// TIA Portal V19 export
FUNCTION "CIP_Filler_512" : Void   // FC98, STL
TITLE = CIP OF FILLING MACHINE
{ S7_Optimized_Access := 'TRUE' }
NAME : CIPTANK
VERSION : 0.0
// Setpoint for Cip forward changed to real from integer
// 
// CIP Program 1 = Rinse-caustic-rinse-acid-rinse-drain
// CIP Program 2 = rinse=caustic-rinse-drain
// 
// If the combi 512 is in fault, the CIP_PUMP_ON input is false, thus M0139 is
// de-engerised and the sequence is held. When the sequence is held steam and 
// chemical valves are de-engerised.
// 
// Version 15 - 25/1/13 ...AFL
// Reset of "M_CAUSTIC_READY" ,"M_RINSE_READY", "M_ACID_READY", in step 1 after 
// occurence of CIP going through without dosing any caustic into CIP solution.
// 
// Version 16 - 22/02/13 ...MC
// In addition to above comment, "CT_LYE_OK", "CT_ACID_OK" also reset in same 
// step.
// stored: AutoNumber false
   VAR_TEMP
      RinseCount : Int;
      Count : Int;
      TEMP0 : Real;
      TEMP2 : Real;
   END_VAR
BEGIN

NETWORK
TITLE = CIP FILLING MACHINE
// Comment
// 
// 
//  Productline being cleaned - Q21.5
      A     "S0 CIP TANK";
      =     "ProdLineBeingCleaned";

// CIP Release - Q21.7
      A     "FS01.81";  // Return flow switch
      A     "Request CIP Pump ON";  //If CIP_PUMP_ON is false
      A(;
      O     "M_CAUSTIC_READY";  //reset CIP release signal
      O     "M_RINSE_READY";
      O     "M_ACID_READY";
      );
      O(;
      A     "Filler_CIP_512_DB".Drain_Ready;  // drain
      A     "Request Drain";
      );
      =     "M_CIP Release";

//   Time Stop - Q21.6
// If a FB error exists sent time stop signal to combi 512
      O     "ItemAlarmsOP".Item[9];  //FB_FAULT_VALVE_01_15
      O     "ItemAlarmsOP".Item[10];  //FB_FAULT_MOTOR_01_39
//  O     "ItemAlarmsOP".FB_FAULT_MOTOR_01_30
      O     "ItemAlarmsOP".Item[12];  //FB_FAULT_VALVE_02_37
      O     "ItemAlarmsOP".Item[13];  //FB_FAULT_VALVE_02_38
      O     "ItemAlarmsOP".Item[14];  //FB_FAULT_VALVE_01_16
      O     "ItemAlarmsOP".Item[15];  //FB_FAULT_VALVE_01_17
//   O     "ItemAlarmsOP".FB_FAULT_VALVE_01_08
//   O     "ItemAlarmsOP".FB_FAULT_VALVE_01_01
//   O     "ItemAlarmsOP".FB_FAULT_VALVE_01_03
//    O     "ItemAlarmsOP".FB_FAULT_VALVE_01_04
//      O     "ItemAlarmsOP".FB_FAULT_VALVE_01_09
//   O     "ItemAlarmsOP".FB_FAULT_VALVE_01_11
      O     "ItemAlarmsOP".Item[6];  //FB_FAULT_VALVE_01_12
      O     "ItemAlarmsOP".Item[7];  //FB_FAULT_VALVE_01_13
      O     "ItemAlarmsOP".Item[8];  //FB_FAULT_VALVE_01_14

//      O     "ItemAlarmsOP".FB_FAULT_VALVE_09_10
//      O     "ItemAlarmsOP".FB_FAULT_VALVE_09_11
//     O     "ItemAlarmsOP".FB_FAULT_VALVE_09_12

//      O     "ItemAlarmsOP".FB_FAULT_VALVE_01_19
      O     "ItemAlarmsOP".Item[18];  //FB_FAULT_VALVE_WATERPUMP
//    O     "ItemAlarmsOP".FB_FAULT_VALVE_09_04
//    O     "ItemAlarmsOP".FB_FAULT_VALVE_09_05
//    O     "ItemAlarmsOP".FB_FAULT_VALVE_09_06
//    O     "ItemAlarmsOP".FB_FAULT_VALVE_09_07
//    O     "ItemAlarmsOP".FB_FAULT_VALVE_09_08
//     O     "ItemAlarmsOP".FB_FAULT_VALVE_09_09
//      =     "M_Time Stop CIP"

      A     "S0 FILLER";
      A     "Combi 512 In USE";
      S     "M_Time Stop CIP";
      R     "LEDAssignment".F12_BUTTON;

      JCN   M03f;
      L     1;  //Display "CIP held Object Error"
      T     "Filler_CIP_512_DB".CIPScreenCenterMessage;
      JU    M040;
M03f: A     "S0 FILLER";
      A     "Combi 512 In USE";
      A     "M_Time Stop CIP";

      JCN   M041;
      L     2;  //Display Press F12 to Resume FILLER CIP
      T     "Filler_CIP_512_DB".CIPScreenCenterMessage;


M041: A     "S0 FILLER";
      A     "Combi 512 In USE";
      A     "M_Time Stop CIP";

      A     "LEDAssignment".F12_BUTTON;
      JCN   M040;

      L     0;  //Clear displayed message
      T     "Filler_CIP_512_DB".CIPScreenCenterMessage;
      R     "M_Time Stop CIP";
      R     "LEDAssignment".F12_BUTTON;




M040: NOP   0;




//*****************

      AN    "Combi 512 In USE";
      BEC;

//Drain Request - aborted cip
      A     "Request Drain";
      A     "S0 FILLER";
      S     "S1 FILLER";
      S     "S2 FILLER";
      S     "S3 FILLER";
      S     "S4 FILLER";
      S     "S5 FILLER";
      S     "S6 FILLER";
      S     "S7 FILLER";
      S     "S8 FILLER";
      S     "S9 FILLER";
      S     "S10 FILLER";
      S     "S11 FILLER";
      S     "S12 FILLER";
      S     "S13 FILLER";
      S     "S14 FILLER";
      S     "S15 FILLER";
      S     "S16 FILLER";
      S     "S17 FILLER";
      S     "S18 FILLER";
      S     "S19 FILLER";
      S     "S20 FILLER";
      S     "S21 FILLER";
      S     "S22 FILLER";
      S     "S23 FILLER";
      S     "S24 FILLER";
      S     "S25 FILLER";
      S     "S26 FILLER";
      S     "S27 FILLER";
      S     "S28 FILLER";
      S     "S29 FILLER";
      S     "S30 FILLER";
      S     "S31 FILLER";
      S     "S32 FILLER";
      S     "S33 FILLER";
      S     "S34 FILLER";
      S     "S35 FILLER";
      S     "S36 FILLER";
      S     "S37 FILLER";
      S     "S38 FILLER";
      S     "S39 FILLER";
      S     "S40 FILLER";
      S     "S41 FILLER";
      S     "S42 FILLER";
      S     "S43 FILLER";
      S     "S44 FILLER";


      AN    "S0 FILLER";
      R     "S1 FILLER";
      R     "S2 FILLER";
      R     "S3 FILLER";
      R     "S4 FILLER";
      R     "S5 FILLER";
      R     "S6 FILLER";
      R     "S7 FILLER";
      R     "S8 FILLER";
      R     "S9 FILLER";
      R     "S10 FILLER";
      R     "S11 FILLER";
      R     "S12 FILLER";
      R     "S13 FILLER";
      R     "S14 FILLER";
      R     "S15 FILLER";
      R     "S16 FILLER";
      R     "S17 FILLER";
      R     "S18 FILLER";
      R     "S19 FILLER";
      R     "S20 FILLER";
      R     "S21 FILLER";
      R     "S22 FILLER";
      R     "S23 FILLER";
      R     "S24 FILLER";
      R     "S25 FILLER";
      R     "S26 FILLER";
      R     "S27 FILLER";
      R     "S28 FILLER";
      R     "S29 FILLER";
      R     "S30 FILLER";
      R     "S31 FILLER";
      R     "S32 FILLER";
      R     "S33 FILLER";
      R     "S34 FILLER";
      R     "S35 FILLER";
      R     "S36 FILLER";
      R     "S37 FILLER";
      R     "S38 FILLER";
      R     "S39 FILLER";
      R     "S40 FILLER";
      R     "S41 FILLER";
      R     "S42 FILLER";
      R     "S43 FILLER";
      R     "S44 FILLER";
      R     "S45 FILLER";
      R     "S46 FILLER";
      R     "S47 FILLER";
      R     "S48 FILLER";
      R     "S49 FILLER";
      BEC;

//    Step 1 Set route for filler
      A     "S1 FILLER";
      JC    M001;
      R     "MM0139";
      S     "MY0114";  // drain
      S     "MY0116";
      S     "MY0117";
//   S     "MY0119"             On Old Comb1 505
      R     "M_RINSE_READY";  //Reset  at start of CIP
      R     "M_CAUSTIC_READY";  //after CIP when throught without
      R     "M_ACID_READY";  //any caustic 25/1/13 ..AFL
      R     "CT_LYE_OK";
      R     "CT_ACID_OK";
      R     "AutoTT0172/IP0157";
      R     "ManTT0172/IP0157";
      S     "S1 FILLER";
      BEU;

//Control heating
M001: A     "B01.42";  // low level in balance tank
      A     "MM0139";  // inhibit heating if off
      A     "ST_HEAT IP0157";
      =     "AutoTT0172/IP0157";
//     =     "Y0158"                   //replaced with new condition, below:

//condition for 01.58 deactivation Measured Temp >= (setpoint + 10 deg C).
      A(;
      A     "B01.42";
      A     "MM0139";
      A     "ST_HEAT IP0157";

      JNB   M042;
      L     "PID_TT0172/IP0157".TT0172SpDBD;
      L     10.0;
      +R;
      T     #TEMP0;
      AN    OV;

      SAVE;
      CLR;
M042: A     BR;
      );
      A(;
      L     "MeasuredValues".TT0172REAL;


      L     #TEMP0;  // low level in balance tank
      <R;  // inhibit heating if off
      );
      =     "Y0158";
      A     "Request CIP Pump ON";
//new condition ends here


//Control CIP PUMP - M0139
      A     "Filler_CIP_512_DB".M0139_db96;
      =     "MM0139";
      A     "MM0139";

//Control lye dosing
      A     "Filler_CIP_512_DB".LyeRequest_db96;
      =     "S.T.01.REQUEST LYE";
      A     "MM0139";

//Control acid dosing
      A     "Filler_CIP_512_DB".AcidReques_db96;
      =     "S.T.01.REQUEST ACID";

NETWORK
TITLE = STEP 02 FILLER
// Comment  Step 2 Wait for route to be ready
      A     "S2 FILLER";
      JC    M002;
      AN    "Y0116S";
      BEC;
      AN    "Y0117S";
      BEC;
//      AN    "Y0119S"
//      BEC
      S     "S2 FILLER";
      BEU;
M002: NOP   0;

NETWORK
TITLE = Prerinse
// Comment  Step 3 Wait for "RINSE REQUEST" signal from filler machine
      A     "S3 FILLER";
      JC    M003;
      AN    "RINSE_REQ";
      BEC;
      S     "CONTROL CIP TANK";
      S     "MY0115";
      S     "S3 FILLER";
      BEU;
M003: NOP   0;

NETWORK
TITLE = Prerinse
// Comment  Step 4 Wait for level in balance tank 01.40
      A     "S4 FILLER";
      JC    M004;
      AN    "B01.41";
      BEC;
      L     "Setpoints".TT01172SpLyeFiller;  // "DB SETPOINTS".TT01172SpLyeFiller
      T     "PID_TT0172/IP0157".TT0172SpDBD;
//      T     "PID_TT0172/IP0157".TT0172SpPID
      S     "ST_HEAT IP0157";
      S     "Filler_CIP_512_DB".M0139_db96;
      S     "S4 FILLER";
      BEU;
M004: NOP   0;

NETWORK
TITLE = Prerinse
// Comment  Step 5 Wait for return flow FS01.81
      A     "S5 FILLER";
      JC    M005;
      AN    "FS01.81";
      BEC;
      S     "TIM19";
      S     "S5 FILLER";
      BEU;
M005: NOP   0;

NETWORK
TITLE = Prerinse
// Comment Step 6 Wait for delay return flow
      A     "S6 FILLER";
      JC    M006;
      A     "Tag_62";
      BEC;
      L     0;
      T     "Filler_CIP_512_DB".Count;
      S     "M_RINSE_READY";
      S     "S6 FILLER";
      BEU;
M006: NOP   0;

NETWORK
TITLE = Prerinse
// Comment Step 7 Wait for prerinse to finished (conroled by filler)
      A     "S7 FILLER";
      JC    M007;
      AN    "RINSE_REQ";
      JC    M032;
      L     0;
      T     "Filler_CIP_512_DB".Count;
M032: AN    "1hz_oneshot_valve handle";
      JC    M033;
      L     "Filler_CIP_512_DB".Count;
      L     1;
      +I;
      T     "Filler_CIP_512_DB".Count;


M033: L     "Filler_CIP_512_DB".Count;
      L     4;
      <I;
      =     "Filler_CIP_512_DB".RequestOffDelay;


      ON    "Request CIP Pump ON";  //HOLD - If CIP_PUMP_ON is false
      O     "RINSE_REQ";  //
      O     "Filler_CIP_512_DB".RequestOffDelay;
      BEC;
      R     "M_RINSE_READY";
//      R     "CONTROL CIP TANK"
//      R     "Y01.15"
      S     "S7 FILLER";
      BEU;
M007: NOP   0;

NETWORK
TITLE = Prerinse
// Comment  Step 8  Wait for low level LSL01.42
      A     "S8 FILLER";
      JC    M008;
//      R     "ST_HEAT IP0157"
//      R     "MM01.39"
      S     "S8 FILLER";
      BEU;
M008: NOP   0;

NETWORK
TITLE = Prerinse
// Comment  Step 9  Dummy
      A     "S9 FILLER";
      JC    M009;
      S     "S9 FILLER";
      BEU;
M009: NOP   0;

NETWORK
TITLE = Caustic
// Comment  Step 10 Wait for "CAUSTIC REQUEST" from filler
      A     "S10 FILLER";
      JC    M00a;
      AN    "CAUSTIC_REQ";
      BEC;
      S     "CONTROL CIP TANK";
      S     "MY0115";
      R     "MY0114";
      S     "S10 FILLER";
      BEU;
M00a: NOP   0;

NETWORK
TITLE = Caustic
// Comment  Step 11 Wait for level in balance tank 01.40
      A     "S11 FILLER";
      JC    M00b;
      ON    "Request CIP Pump ON";  // hold sequence if false
      ON    "B01.42";
      BEC;
      S     "ST_HEAT IP0157";
      S     "Filler_CIP_512_DB".M0139_db96;
      S     "S11 FILLER";
      BEU;
M00b: NOP   0;

NETWORK
TITLE = Caustic
// Comment Step 12 Wait for return flow FS01.81
      A     "S12 FILLER";
      JC    M00c;
      AN    "FS01.81";
      BEC;
      S     "Filler_CIP_512_DB".LyeRequest_db96;
      S     "S12 FILLER";
      BEU;
M00c: NOP   0;

NETWORK
TITLE = Caustic
// Comment  Step 13  Wait for min lye concentration return (Not used)
      A     "S13 FILLER";
      JC    M00d;
      S     "S13 FILLER";
      BEU;
M00d: NOP   0;

NETWORK
TITLE = Caustic
// Comment  Step 14 Wait for caustic concentration to be OK
      A     "S14 FILLER";
      JC    M00e;
      AN    "CT_LYE_OK";
      BEC;
      R     "Filler_CIP_512_DB".LyeRequest_db96;
      R     "CT_LYE_OK";
      S     "S14 FILLER";
      BEU;
M00e: NOP   0;

NETWORK
TITLE = Caustic
// Comment  Step 15 Wait for temperature to be OK
      A     "S15 FILLER";
      JC    M00f;
      L     "MeasuredValues".TT0180REAL;  // "DB-ANALOG INPUT".TT0180MEAS
      L     "Setpoints".MinCipFillerTempTT01;  //"DB SETPOINTS".MinCipFillerTempTT01
      <R;
      BEC;
      L     0;
      T     "Filler_CIP_512_DB".Count;
      S     "M_CAUSTIC_READY";
      S     "S15 FILLER";
      BEU;
M00f: NOP   0;

NETWORK
TITLE = Caustic
// Comment  Step 16 Wait for caustic to be finished (controled by filler)
      A     "S16 FILLER";
      JC    M010;
      AN    "CAUSTIC_REQ";
      JC    M034;
      L     0;
      T     "Filler_CIP_512_DB".Count;
M034: AN    "1hz_oneshot_valve handle";
      JC    M035;
      L     "Filler_CIP_512_DB".Count;
      L     1;
      +I;
      T     "Filler_CIP_512_DB".Count;


M035: L     "Filler_CIP_512_DB".Count;
      L     4;
      <I;
      =     "Filler_CIP_512_DB".RequestOffDelay;

      ON    "Request CIP Pump ON";  // hold sequence if false
      O     "CAUSTIC_REQ";
      O     "Filler_CIP_512_DB".RequestOffDelay;
      BEC;
      R     "M_CAUSTIC_READY";
      S     "MY0114";
      S     "S16 FILLER";
      BEU;
M010: NOP   0;

NETWORK
TITLE = Caustic
// Comment  Step 17 Wait for min lye concentration return
      A     "S17 FILLER";
      JC    M011;
//      R     "CONTROL CIP TANK"
      S     "S17 FILLER";
      BEU;
M011: NOP   0;

NETWORK
TITLE = Caustic
// Comment  Step 18  Wait for low level in balance tank LSL01.42
      A     "S18 FILLER";
      JC    M012;
//      A     "B01.42"
//      BEC
//      R     "ST_HEAT IP0157"
//      R     "MM01.39"
      S     "S18 FILLER";
      BEU;
M012: NOP   0;

NETWORK
TITLE = Caustic
// Comment  Step 19 Check which CIP program selected 
// 
// If Program 1 is Selected both "PROG_1_SELECTED" and "PROG_2_SELECTED" are true
// If Program 2 is Selected "PROG_1_SELECTED" is FALSE and "PROG_2_SELECTED" is 
// TRUE
      A     "S19 FILLER";
      JC    M013;
      A     "PROG_1_SELECTED";  // Rinse - Caustic  -   Middle rinse - Acid - Final Rinse - Drain  Prog 1
      A     "PROG_2_SELECTED";  // Rinse - Caustic  -   Final rinse - Drain  Prog 2
      JC    M03e;
      S     "S19 FILLER";
      S     "S20 FILLER";
      S     "S21 FILLER";
      S     "S22 FILLER";
      S     "S23 FILLER";
      S     "S24 FILLER";
      S     "S25 FILLER";
      S     "S26 FILLER";
      S     "S27 FILLER";
      S     "S28 FILLER";
      S     "S29 FILLER";
      S     "S30 FILLER";
      S     "S31 FILLER";
      S     "S30 FILLER";
      S     "S32 FILLER";
      S     "S33 FILLER";
      S     "S34 FILLER";
      S     "S35 FILLER";
      S     "S36 FILLER";
      S     "S37 FILLER";
      S     "S38 FILLER";
      S     "S39 FILLER";
      S     "S40 FILLER";
      BEC;
M03e: SET;
      S     "S19 FILLER";
      BEU;
M013: NOP   0;

NETWORK
TITLE = Middle rinse
// Comment  Step 20 Wait for "RINSE REQUEST" from filler
      A     "S20 FILLER";
      JC    M014;
      AN    "RINSE_REQ";
      BEC;
      L     25.0;
      T     "PID_TT0172/IP0157".TT0172SpDBD;
//      T     "PID_TT0172/IP0157".TT0172SpPID
      S     "MY0114";
      S     "CONTROL CIP TANK";
      S     "MY0115";
      S     "S20 FILLER";
      BEU;
M014: NOP   0;

NETWORK
TITLE = Middle rinse
// Comment  Step 21 Wait for level in balance tank
      A     "S21 FILLER";
      JC    M015;
      AN    "B01.42";
      BEC;
      S     "ST_HEAT IP0157";
      S     "Filler_CIP_512_DB".M0139_db96;
      S     "S21 FILLER";
      BEU;
M015: NOP   0;

NETWORK
TITLE = Middle rinse
// Comment  Step 22 Wait for return flow FS01.81
      A     "S22 FILLER";
      JC    M016;
      AN    "FS01.81";
      BEC;
      S     "S22 FILLER";
      BEU;
M016: NOP   0;

NETWORK
TITLE = Middle rinse
// Comment  Step 23 Wait for temperature to be OK
      A     "S23 FILLER";
      JC    M017;
      L     "MeasuredValues".CT0182REAL;  // "DB-ANALOG INPUT".CT0182REAL
      L     5.0;
      >=R;
      BEC;
      S     "M_RINSE_READY";
      S     "S23 FILLER";
      BEU;
M017: NOP   0;

NETWORK
TITLE = Middle rinse
// Comment  Step 24 Wait for middle rinse to finished (controled by filler)
      A     "S24 FILLER";
      JC    M018;
      AN    "RINSE_REQ";
      JC    M036;
      L     0;
      T     "Filler_CIP_512_DB".Count;
M036: AN    "1hz_oneshot_valve handle";
      JC    M037;
      L     "Filler_CIP_512_DB".Count;
      L     1;
      +I;
      T     "Filler_CIP_512_DB".Count;


M037: L     "Filler_CIP_512_DB".Count;
      L     4;
      <I;
      =     "Filler_CIP_512_DB".RequestOffDelay;

      ON    "Request CIP Pump ON";  // hold sequence if false
      O     "RINSE_REQ";  // Hold count
      O     "Filler_CIP_512_DB".RequestOffDelay;
      BEC;
      R     "M_RINSE_READY";
//      R     "CONTROL CIP TANK"
//      R     "MY01.15"
      R     "MY0114";
      S     "S24 FILLER";
      BEU;
M018: NOP   0;

NETWORK
TITLE = Middle rinse
// Comment  Step 25 Wait for low level in balance tank LSL01.42
      A     "S25 FILLER";
      JC    M019;
//      A     "B01.42"
//      BEC
//      R     "ST_HEAT IP0157"
//      R     "MM01.39"
      S     "S25 FILLER";
      BEU;
M019: NOP   0;

NETWORK
TITLE = Middle rinse
// Comment  Step 26 (Not used)
      A     "S26 FILLER";
      JC    M01a;
      S     "S26 FILLER";
      BEU;
M01a: NOP   0;

NETWORK
TITLE = Middle rinse
// Comment  Step 27 (Not used)
      A     "S27 FILLER";
      JC    M01b;
      S     "S27 FILLER";
      BEU;
M01b: NOP   0;

NETWORK
TITLE = Middle rinse
// Comment  Step 28 (Not used)
      A     "S28 FILLER";
      JC    M01c;
      S     "S28 FILLER";
      BEU;
M01c: NOP   0;

NETWORK
TITLE = Middle rinse
// Comment  Step 29 (Not used)
      A     "S29 FILLER";
      JC    M01d;
      S     "S29 FILLER";
      BEU;
M01d: NOP   0;

NETWORK
TITLE = Acid
// Comment  Step 30 Wait for "ACID REQUEST" from filler
      A     "S30 FILLER";
      JC    M01e;
      AN    "ACID_REQ";
      BEC;
      L     "Setpoints".TT01172SpAcidFiller;  //"DB SETPOINTS".TT01172SpAcidFiller
      T     "PID_TT0172/IP0157".TT0172SpDBD;
      S     "CONTROL CIP TANK";
      S     "MY0115";
      S     "S30 FILLER";
      BEU;
M01e: NOP   0;

NETWORK
TITLE = Acid
// Comment  Step 31 Wait for level in balance tank
      A     "S31 FILLER";
      JC    M01f;
      AN    "B01.42";
      BEC;
      S     "ST_HEAT IP0157";
      S     "Filler_CIP_512_DB".M0139_db96;
      S     "S31 FILLER";
      BEU;
M01f: NOP   0;

NETWORK
TITLE = Acid
// Comment  Step 32 Wait for renturn flow FS01.81
      A     "S32 FILLER";
      JC    M020;
      AN    "FS01.81";
      BEC;
      S     "Filler_CIP_512_DB".AcidReques_db96;
      R     "MY0114";
      S     "S32 FILLER";
      BEU;
M020: NOP   0;

NETWORK
TITLE = Acid
// Comment  Step 33 Wait for min acid concentration reurn
      A     "S33 FILLER";
      JC    M021;
      S     "S33 FILLER";
      BEU;
M021: NOP   0;

NETWORK
TITLE = Acid
// Comment  Step 34 Wait for acid concentration to be OK
      A     "S34 FILLER";
      JC    M022;
      AN    "CT_ACID_OK";
      BEC;
      R     "Filler_CIP_512_DB".AcidReques_db96;
      R     "CT_ACID_OK";
      S     "S34 FILLER";
      BEU;
M022: NOP   0;

NETWORK
TITLE = Acid
// Comment  Step 35 Wait for temperature to be OK
      A     "S35 FILLER";
      JC    M023;
      L     "MeasuredValues".TT0180REAL;  //"DB-ANALOG INPUT".TT0180MEAS
      L     "Setpoints".MinCipFillerTempTT01;  //"DB SETPOINTS".MinCipFillerTempTT01
      <R;
      BEC;
      S     "M_ACID_READY";
      S     "S35 FILLER";
      BEU;
M023: NOP   0;

NETWORK
TITLE = Acid
// Comment  Step 36 Wait for acid to be finished (controled by filler)
      A     "S36 FILLER";
      JC    M024;
      AN    "ACID_REQ";
      JC    M039;
      L     0;
      T     "Filler_CIP_512_DB".Count;
M039: AN    "1hz_oneshot_valve handle";
      JC    M038;
      L     "Filler_CIP_512_DB".Count;
      L     1;
      +I;
      T     "Filler_CIP_512_DB".Count;


M038: L     "Filler_CIP_512_DB".Count;
      L     4;
      <I;
      =     "Filler_CIP_512_DB".RequestOffDelay;

      ON    "Request CIP Pump ON";  // hold sequence if false
      O     "ACID_REQ";
      O     "Filler_CIP_512_DB".RequestOffDelay;
      BEC;
      R     "M_ACID_READY";
      S     "MY0114";
      L     25.0;
      T     "PID_TT0172/IP0157".TT0172SpDBD;
//      T     "PID_TT0172/IP0157".TT0172SpPID
      S     "S36 FILLER";
      BEU;
M024: NOP   0;

NETWORK
TITLE = Acid
// Comment  Step 37 Wait for min acid concentration return
      A     "S37 FILLER";
      JC    M025;
//      R     "CONTROL CIP TANK"
      S     "S37 FILLER";
      BEU;
M025: NOP   0;

NETWORK
TITLE = Acid
// Comment  Step 38  Wait for low level in balance tank LSL01.42
      A     "S38 FILLER";
      JC    M026;
//      A     "B01.42"
//      BEC
//      R     "ST_HEAT IP0157"
//      R     "MM01.39"
      S     "S38 FILLER";
      BEU;
M026: NOP   0;

NETWORK
TITLE = Acid
// Comment  Step 39 Dummy
      A     "S39 FILLER";
      JC    M027;
      S     "S39 FILLER";
      BEU;
M027: NOP   0;

NETWORK
TITLE = Final rinse
// Comment  Step 40 Wait for "RINSE REQUEST" from filler
      A     "S40 FILLER";
      JC    M028;
      AN    "RINSE_REQ";
      BEC;
      S     "MY0114";
      S     "CONTROL CIP TANK";
      S     "MY0115";
      S     "S40 FILLER";
      BEU;
M028: NOP   0;

NETWORK
TITLE = Final rinse
// Comment  Step 41 Wait for level in balance tank
      A     "S41 FILLER";
      JC    M029;
      AN    "B01.42";
      BEC;
      S     "ST_HEAT IP0157";
      S     "Filler_CIP_512_DB".M0139_db96;
      S     "S41 FILLER";
      BEU;
M029: NOP   0;

NETWORK
TITLE = Final rinse
// Comment  Step 42 Wait for return flow FS01.81
      A     "S42 FILLER";
      JC    M02a;
      AN    "FS01.81";
      BEC;
      S     "S42 FILLER";
      BEU;
M02a: NOP   0;

NETWORK
TITLE = Final rinse
// Comment  Step 43 Wait for temperature to be OK
      A     "S43 FILLER";
      JC    M02b;
      L     "MeasuredValues".CT0182REAL;  //"DB-ANALOG INPUT".CT0182REAL
      L     5.0;
      >=R;
      BEC;
      L     0;
      T     "Filler_CIP_512_DB".Count;
      S     "M_RINSE_READY";
      S     "S43 FILLER";
      BEU;
M02b: NOP   0;

NETWORK
TITLE = Final rinse
// Comment  Step 44 Wait for Final rinse to finished (controled by filler)
      A     "S44 FILLER";
      JC    M02c;
      AN    "RINSE_REQ";
      JC    M03a;
      L     0;
      T     "Filler_CIP_512_DB".Count;
M03a: AN    "1hz_oneshot_valve handle";
      JC    M03b;
      L     "Filler_CIP_512_DB".Count;
      L     1;
      +I;
      T     "Filler_CIP_512_DB".Count;


M03b: L     "Filler_CIP_512_DB".Count;
      L     4;
      <I;
      =     "Filler_CIP_512_DB".RequestOffDelay;

      ON    "Request CIP Pump ON";  // hold sequence if false
      O     "RINSE_REQ";
      O     "Filler_CIP_512_DB".RequestOffDelay;
      BEC;
      R     "M_RINSE_READY";
//      R     "CONTROL CIP TANK"
//      S     "MY01.14"
      S     "S44 FILLER";
      BEU;
M02c: NOP   0;

NETWORK
TITLE = Final rinse
// Comment  Step 45 Stop Heating and M0139
      A     "S45 FILLER";
      JC    M02d;
      L     0;
      T     "Filler_CIP_512_DB".Count;
      S     "S45 FILLER";
      BEU;
M02d: NOP   0;

NETWORK
TITLE = Final rinse
// Comment  Step 46 Wait for drain Request
// 
// Delay drain ready signal for time
      A     "S46 FILLER";
      JC    M02e;
// Delay Drain Ready signal for 4 seconds
//      A     "Drain Request"
//      AN    "1hz_oneshot_valve handle"
//      JC    t017
//      L     "Filler_CIP_512_DB".Count
//      L     1
//      +I
//      T     "Filler_CIP_512_DB".Count

//t017: L     "Filler_CIP_512_DB".Count   // Delay Drain Ready signal for 4 seconds
//      L     4                           //
//      <I


      AN    "Request Drain";
      BEC;
      R     "CONTROL CIP TANK";
      S     "MY0114";
      S     "MY0116";
      R     "Filler_CIP_512_DB".LyeRequest_db96;
      R     "Filler_CIP_512_DB".AcidReques_db96;
      R     "M_RINSE_READY";
      R     "M_CAUSTIC_READY";
      R     "M_ACID_READY";
      R     "RINSE_READY";
      R     "CAUSTIC_READY";
      R     "ACID_READY";
      R     "ST_HEAT IP0157";
      R     "Filler_CIP_512_DB".M0139_db96;


      S     "S46 FILLER";
      BEU;
M02e: NOP   0;

NETWORK
TITLE = Final rinse
// Comment  Step 47 Wait for valve and motor status
      A     "S47 FILLER";
      JC    M02f;
      O     "M0139S";
      ON    "Y0114S";
      ON    "Y0116S";
      BEC;
      AN    "1hz_oneshot_valve handle";
      JC    M03c;
      L     "Filler_CIP_512_DB".Count;
      L     1;
      +I;
      T     "Filler_CIP_512_DB".Count;
M03c: L     "Filler_CIP_512_DB".Count;  // Delay Drain Ready signal for 20 seconds
      L     20;  //
      <I;
      S     "Filler_CIP_512_DB".Drain_Ready;
      S     "S47 FILLER";
      L     0;
      T     "Filler_CIP_512_DB".Count;
      BEU;
M02f: NOP   0;

NETWORK
TITLE = Final rinse
// Comment  Step 48 Wait for drain request = false
      A     "S48 FILLER";
      JC    M030;
      AN    "Request Drain";
      JC    M03d;
      AN    "1hz_oneshot_valve handle";
      JC    M03d;
      L     "Filler_CIP_512_DB".Count;
      L     1;
      +I;
      T     "Filler_CIP_512_DB".Count;

M03d: L     "Filler_CIP_512_DB".Count;  // Delay Drain Ready signal for 4 seconds
      L     220;  //
      <I;
      AN    "Continue_in program";  //Get out clause if 512 finishes before Count=>220
      BEC;
      A     "Request Drain";
      BEC;
      R     "Continue_in program";
      R     "Filler_CIP_512_DB".Drain_Ready;
      R     "MY0114";
      S     "S48 FILLER";
      BEU;
M030: NOP   0;

NETWORK
TITLE = Final rinse
// Comment  Step 49 CIP Finished
      A     "S49 FILLER";
      JC    M031;
      S     "S49 FILLER";
      R     "S0 FILLER";
      R     "LEDAssignment".K9_FLASH;  // "FLASH_K9_CIP_FIL"
      R     "LEDAssignment".K9_LIGHT;  // "LIGHT_K9_CIP_FIL"
      R     "AutoTT0172/IP0157";
      R     "Filler_CIP_512_DB".M0139_db96;
      R     "MY0114";  // drain
      R     "MY0115";
      R     "MY0116";
      R     "MY0117";
//    R     "MY0119"

      BEU;
M031: NOP   0;
END_FUNCTION
